FUNCTION_BLOCK SkillNeu EXTENDS SkillBAsisGeruest
VAR_INPUT
	b_Test			:BOOL;
END_VAR
VAR_OUTPUT
END_VAR
VAR
END_VAR

END_FUNCTION_BLOCK

(* stored: Version 1.1.0.1
   POU SkillNeu: Id {2cead17c-3d2a-4594-834a-efc0218ed1e6}, SpecialFunc None *)
